# EPICS autosave request: 3-0/iocBoot/iocGalil/galilTestApp_positions.req
$(P)A.DVAL
$(P)B.DVAL
$(P)C.DVAL
$(P)D.DVAL
$(P)E.DVAL
$(P)F.DVAL
$(P)G.DVAL
$(P)H.DVAL
